// TwinCAT 3 PLC project Gemma
// ProgramVersion: 3.1.4024.0
// libraries:
//   CmpBitmapPool, * (System)
//   Tc2_Standard, * (Beckhoff Automation GmbH)
//   Tc2_System, * (Beckhoff Automation GmbH)
//   Tc3_Module, * (Beckhoff Automation GmbH)
//   VisuDialogs, * (System)
// project tree:
//   DUTs/ E_GEMMA.TcDUT (not stored)
//   / GlobalTextList.TcGTLO, PlcTask.TcTTO, Visualization Manager.TcVMO (not stored)
//   POUs/Estacion/ FB_Coordinador_SFC.TcPOU (not stored), FB_Director.TcPOU (not stored), FB_Estacion.TcPOU
//   POUs/ MAIN.TcPOU
//   POUs/Reloj/ FB_Clock.TcPOU (not stored)
//   POUs/Tareas/ FB_AlimentadorVerificadorDesplazador_SFC.TcPOU (not stored), FB_CheckMaterial_SFC.TcPOU (not stored), FB_Descargador_SFC.TcPOU (not stored), FB_EstacionFinalizar_SFC.TcPOU, FB_EstacionPreparar_SFC.TcPOU (not stored), FB_Rechazador_SFC.TcPOU, FB_ResetDescargador_SFC.TcPOU, FB_SituarPale_SFC.TcPOU (not stored), FB_TransferirPale_SFC.TcPOU
//   VISUs/ ImagePool.TcIPO (not stored), Visualization.TcVIS
// (motion and I/O tree: see PLC project manual)
// real-time tasks:
//   TASK PlcTask: cycle T#10ms, priority 20, ADS port 350
//   TASK PlcTask1: cycle T#10ms, priority 21, ADS port 351
// variable links:
//   Gemma/Gemma Instance <-> Device 1 (EtherCAT)/Term 1 (EK1200)/Term 2 (EL1008)
//     PlcTask Inputs/MAIN.Estacion.Codigo_pale_bit_0 <-> Channel 7/Codigo de palé bit 0
//     PlcTask Inputs/MAIN.Estacion.Codigo_pale_bit_1 <-> Channel 8/Codigo de palé bit 1
//     PlcTask Inputs/MAIN.Estacion.EstacionConectada <-> Channel 5/Parte operativa conectada (armada)
//     PlcTask Inputs/MAIN.Estacion.Presencia_pale <-> Channel 6/presencia de palé
//     PlcTask Inputs/MAIN.Estacion.Pulsador_marcha <-> Channel 3/Pulsador de marcha
//     PlcTask Inputs/MAIN.Estacion.Pulsador_parada_NC <-> Channel 4/Pulsador de parada [NC]
//     PlcTask Inputs/MAIN.Estacion.Pulsador_parada_emergencia <-> Channel 1/Pulsador de parada de emergencia
//     PlcTask Inputs/MAIN.Estacion.Selector_modo_manual <-> Channel 2/Selector de modo manual
//   Gemma/Gemma Instance <-> Device 1 (EtherCAT)/Term 1 (EK1200)/Term 3 (EL1008)
//     PlcTask Inputs/MAIN.Estacion.Codigo_pale_bit_2 <-> Channel 1/Código de palé bit 2
//     PlcTask Inputs/MAIN.Estacion.Detector_presion <-> Channel 2/Detector de presión
//   Gemma/Gemma Instance <-> Device 1 (EtherCAT)/Term 1 (EK1200)/Term 6 (EL1008)
//     PlcTask Inputs/MAIN.Estacion.Desplazador_detras <-> Channel 7/Cilindro del desplazador detrás
//     PlcTask Inputs/MAIN.Estacion.Horizontal_descargador_delante <-> Channel 2/Cilindro horizontal del descargador delante (sobre el palé)
//     PlcTask Inputs/MAIN.Estacion.Horizontal_descargador_detras <-> Channel 1/Cilindro horizontal del descargador detrás (sobre el punto de descarga)
//     PlcTask Inputs/MAIN.Estacion.Verificador_abajo <-> Channel 6/Cilindro del verificador abajo
//     PlcTask Inputs/MAIN.Estacion.Verificador_arriba <-> Channel 5/Cilindro del verificador arriba
//     PlcTask Inputs/MAIN.Estacion.Vertical_descargador_abajo <-> Channel 4/Cilindro vertical del descargador abajo
//     PlcTask Inputs/MAIN.Estacion.Vertical_descargador_arriba <-> Channel 3/Cilindro vertical del descargador arriba
//   Gemma/Gemma Instance <-> Device 1 (EtherCAT)/Term 1 (EK1200)/Term 7 (EL1008)
//     PlcTask Inputs/MAIN.Estacion.Base_en_alimentador <-> Channel 3/Presencia de base en el alimentador

CONFIGURATION Gemma
    RESOURCE PLC ON TwinCAT3
        TASK PlcTask(INTERVAL := T#10ms, PRIORITY := 20);
        PROGRAM MAIN WITH PlcTask : MAIN;
    END_RESOURCE
END_CONFIGURATION

// ---- POUs/MAIN.TcPOU
PROGRAM MAIN
VAR
	
	//Pulsador AT %I*: BOOL;
	//Lampara AT %Q*: BOOL;
	
	Estacion: FB_Estacion;

END_VAR

Estacion();

END_PROGRAM

// ---- POUs/Estacion/FB_Estacion.TcPOU
FUNCTION_BLOCK FB_Estacion
VAR_INPUT
    EstadoPausa: BOOL;
    EstadoReinicia: BOOL;
    CiclosSolicitados: UINT := 0;
    
    Tcheck: TIME := T#1S;
    Treset: TIME := T#1S;
    Tdesplazador: TIME := T#1S;
	Tcinta: TIME := T#0.5S;
END_VAR
VAR_OUTPUT
    CondicionInicial: BOOL := TRUE;
    CiclosPendientes: UINT;
    CiclosAceptados: UINT;
	CiclosRechazados: UINT;
    PaleCodigo: BYTE;
	pieza_ok: BOOL;
    
    // Entradas comunes
	Base_en_alimentador AT %I*: BOOL;
    Pulsador_parada_emergencia AT %I*: BOOL;
    Selector_modo_manual AT %I*: BOOL;
    Pulsador_marcha AT %I*: BOOL;
    Pulsador_parada_NC AT %I*: BOOL := TRUE; // Contacto normalmente cerrado
    EstacionConectada AT %I*: BOOL := TRUE;
    Detector_presion AT %I*: BOOL := TRUE;

    Presencia_pale AT %I*: BOOL;
    Codigo_pale_bit_0 AT %I*: BOOL;
    Codigo_pale_bit_1 AT %I*: BOOL;
    Codigo_pale_bit_2 AT %I*: BOOL;

    // Entradas espeficicas
    //Terminal 6
	Horizontal_descargador_detras AT %I*: BOOL;
	Horizontal_descargador_delante AT %I*: BOOL;
	Vertical_descargador_arriba AT %I*: BOOL;
	Vertical_descargador_abajo AT %I*: BOOL;
	Verificador_arriba AT %I*: BOOL;
	Verificador_abajo AT %I*: BOOL;
	Desplazador_detras AT %I*: BOOL;
	//Desplazador_delante AT %I*: BOOL;
	Alimentador_detras AT %I*: BOOL;
	
	
	//Terminal 7
	Alimentador_delante AT %I*: BOOL;
	Vacio_obtenido_vacuostato_descargador AT %I*: BOOL;

END_VAR
VAR
	ModoAnterior: E_GEMMA;    

    // Bloques funcionales
    CLK: FB_Clock;	

    // Bloques funcionales
	Director : FB_Director;
    Coordinador: FB_Coordinador_SFC;
	ChequeaMaterial: FB_CheckMaterial_SFC;
	AlimentadorVerificadorDesplazador: FB_AlimentadorVerificadorDesplazador_SFC;
    SituarPale: FB_SituarPale_SFC;
	ResetDescargador: FB_ResetDescargador_SFC;
    Descargador: FB_Descargador_SFC;
    Rechazador: FB_Rechazador_SFC;
    TransferirPale: FB_TransferirPale_SFC;
	Finalizar: FB_EstacionFinalizar_SFC;
	Preparar: FB_EstacionPreparar_SFC;
    
    // Salidas comunes
    Desconecta_parte_operativa AT %Q*: BOOL;
    Lampara_falta_material AT %Q*: BOOL;
    Lampara_marcha AT %Q*: BOOL;
    Lampara_alarma AT %Q*: BOOL;

    Activa_marcha_motor_cinta AT %Q*: BOOL;
    Invierte_marcha_motor_cinta AT %Q*: BOOL;
    Retenedor_pale_baja AT %Q*: BOOL;
    Separador_pale_sube AT %Q*: BOOL;
    
    //Terminal 8
	Descargador_adelante AT %Q*: BOOL;
	Descargador_atras AT %Q*: BOOL;
	Descargador_baja AT %Q*: BOOL;
	Rechazador_adelante AT %Q*: BOOL;
	Verificador_baja AT %Q*: BOOL;
	Desplazador_adelante AT %Q*: BOOL;
	Alimentador_adelante AT %Q*: BOOL;
	Eyector_succiona AT %Q*: BOOL;
	SFCPause: BOOL;
END_VAR

// Modo Automático
//IF NOT Selector_Modo_Manual THEN
CLK();

    // Bloques Funcionales
    Director(
        CondicionInicial := CondicionInicial,
        CondicionMarcha:= (CiclosSolicitados > 0) AND CondicionInicial,
        Emergencia := Pulsador_parada_emergencia,
        Finalizada := Finalizar.Done,
        FinTarea := (CiclosPendientes = 0),
        FinCiclo := Coordinador.Done,
        Manual := Selector_modo_manual,
        Marcha := Pulsador_marcha,
        ParaCiclo := NOT Pulsador_parada_NC,
        Preparada := Preparar.Done,
        Reinicia := EstadoReinicia
    );
	
	IF (Director.Modo <> E_GEMMA.F4) THEN

    SituarPale( //SituarPale
        SFCPause := NOT EstadoReinicia AND EstadoPausa,
        SFCReset := EstadoReinicia,
        Ack := NOT Coordinador.SituaPale,
        Execute := Coordinador.SituaPale,
        Tcinta := Tcinta,
        Presencia_pale := Presencia_pale,
           //Codigo_pale_bit_0 := Codigo_pale_bit_0,
        //Codigo_pale_bit_1 := Codigo_pale_bit_1,
        //Codigo_pale_bit_2 := Codigo_pale_bit_2

    );

	// Bloques Funcionales
	Coordinador(

		CiclosPendientes := CiclosPendientes,
		CiclosAceptados := CiclosAceptados,
		CiclosSolicitados := CiclosSolicitados,
		CiclosRechazados := CiclosRechazados,
		SFCPause := NOT EstadoReinicia AND EstadoPausa,
        SFCReset := EstadoReinicia,
		Ack := TRUE,
        Execute := (Director.Modo = E_GEMMA.F1),
		PaleSituado := SituarPale.Done,
		HayMaterial := ChequeaMaterial.Done,
		Verificado := AlimentadorVerificadorDesplazador.Done,
		DescargadorReseteado := ResetDescargador.Done,
        Rechazado := Rechazador.Done,
		BaseCargada := Descargador.Done,
		PaleTransferido := TransferirPale.Done,
		pieza_ok := pieza_ok
		
	);
	
	Preparar(
		
		SFCPause := NOT EstadoReinicia AND EstadoPausa,
        SFCReset := EstadoReinicia,
        Ack := (Director.Modo <> E_GEMMA.F2),
        Execute := (Director.Modo = E_GEMMA.F2),
		Horizontal_descargador_detras := Horizontal_descargador_detras,
		Vertical_descargador_arriba := Vertical_descargador_arriba,
		Presencia_pale := Presencia_pale
	
	);
	
	Finalizar(
		
		SFCPause := NOT EstadoReinicia AND EstadoPausa,
        SFCReset := EstadoReinicia,
        Ack := (Director.Modo <> E_GEMMA.F3),
        Execute := (Director.Modo = E_GEMMA.F3),
		Horizontal_descargador_detras := Horizontal_descargador_detras,
		Vertical_descargador_arriba := Vertical_descargador_arriba,
		Presencia_pale := Presencia_pale
	
	);
	
	SituarPale(

		SFCPause := NOT EstadoReinicia AND EstadoPausa,
        SFCReset := EstadoReinicia,
        Ack := NOT Coordinador.SituaPale,
        Execute := Coordinador.SituaPale,
        Tcinta := Tcinta,
        Presencia_pale := Presencia_pale,
       	//Codigo_pale_bit_0 := Codigo_pale_bit_0,
        //Codigo_pale_bit_1 := Codigo_pale_bit_1,
        //Codigo_pale_bit_2 := Codigo_pale_bit_2

	);
	
	ChequeaMaterial(
		Ack := NOT Coordinador.ChequeaMaterial,
		SFCPause := NOT EstadoReinicia AND EstadoPausa,
        SFCReset := EstadoReinicia,
		Execute := Coordinador.ChequeaMaterial,
		Base_en_Alimentador := Base_en_alimentador,
		Pulsador_marcha := Pulsador_marcha
	);
	
	AlimentadorVerificadorDesplazador(
		
		Ack := NOT Coordinador.VerificaBase,
        Tcheck := Tcheck,
		SFCPause := NOT EstadoReinicia AND EstadoPausa,
        SFCReset := EstadoReinicia,
		Execute := Coordinador.VerificaBase,
		Alimentador_delante := Alimentador_delante,
		Alimentador_detras := Alimentador_detras,
		Verificador_arriba := Verificador_arriba ,
		Verificador_abajo := Verificador_abajo,
		Desplazador_delante := Desplazador_delante,
		Desplazador_detras := Desplazador_detras, 
		
	);
	
	ResetDescargador(

		Ack := NOT Coordinador.ResetDescargador,
		SFCPause := NOT EstadoReinicia AND EstadoPausa,
        SFCReset := EstadoReinicia,
		Execute := Coordinador.ResetDescargador,
		Horizontal_descargador_detras := Horizontal_descargador_detras,
		Vertical_descargador_arriba := Vertical_descargador_arriba
	);
	
	Descargador(
		
		Ack := NOT Coordinador.CargaBase,
		SFCPause := NOT EstadoReinicia AND EstadoPausa,
        SFCReset := EstadoReinicia,
		Execute := Coordinador.CargaBase,
		Horizontal_descargador_detras := Horizontal_descargador_detras,
		Vertical_descargador_abajo := Vertical_descargador_abajo,
		Vacio_obtenido_vacuostato_descargador := Vacio_obtenido_vacuostato_descargador ,
		Vertical_descargador_arriba := Vertical_descargador_arriba ,
		Horizontal_descargador_delante := Horizontal_descargador_delante ,
	
	);	
		
	Rechazador(
		
		Ack := NOT Coordinador.RechazaBase,
		SFCPause := NOT EstadoReinicia AND EstadoPausa,
        SFCReset := EstadoReinicia,
		Execute := Coordinador.RechazaBase,
		Verificador_abajo := Verificador_abajo
		
	);
	
	TransferirPale(
	
		Ack := NOT Coordinador.TransfierePale,
		SFCPause := NOT EstadoReinicia AND EstadoPausa,
        SFCReset := EstadoReinicia,
		Execute := Coordinador.TransfierePale,

	);
	
	//Acciones Comunes
	// Parametros de Salida
	//Lampara_falta_material := ChequeaMaterial.Lampara_falta_material;
	Activa_marcha_motor_cinta := SituarPale.Activa_marcha_motor_cinta OR TransferirPale.Activa_marcha_motor_cinta OR Preparar.Activa_marcha_motor_cinta OR Finalizar.Activa_marcha_motor_cinta;
	//CheckMaterial
	Lampara_alarma := ChequeaMaterial.LamparaAlarma;
	Lampara_falta_material := ChequeaMaterial.Lampara_falta_material;
	//TranferirPale
	 Retenedor_pale_baja := TransferirPale.Retenedor_pale_baja;
	 Separador_pale_sube := TransferirPale.Separador_pale_sube;
	//AlimentadorVerificadorDesplazador
	Alimentador_adelante := AlimentadorVerificadorDesplazador.Alimentador_adelante;
	Verificador_baja := AlimentadorVerificadorDesplazador.Verificador_baja;
	Desplazador_adelante := AlimentadorVerificadorDesplazador.Desplazador_adelante;
	pieza_ok := AlimentadorVerificadorDesplazador.pieza_ok;
	//Descargador
	Eyector_succiona := Descargador.Eyector_succiona;
	Descargador_adelante := Descargador.Descargador_adelante;
	Descargador_atras := Descargador.Descargador_atras OR ResetDescargador.Descargador_atras;
	Descargador_baja := Descargador.Descargador_baja;
	//Rechazador
	Rechazador_adelante := Rechazador.Rechazador_adelante;
	
	IF NOT EstadoPausa THEN
	
		EstadoPausa := not Pulsador_parada_NC;
	
	ELSE
	
		EstadoPausa := NOT Pulsador_marcha;
	
	END_IF

END_IF	
	
// Parametros de Salida
CondicionInicial := EstacionConectada; //AND Desplazador_detras AND Verificador_arriba AND Vertical_descargador_arriba AND Alimentador_detras;

//al iniciar una tarea
IF ((ModoAnterior = E_GEMMA.A1) AND (Director.Modo <> E_GEMMA.A1) AND (CiclosPendientes = 0)) THEN
    CiclosPendientes := CiclosSolicitados;
END_IF

//IF (Director.Modo <> E_GEMMA.F4) THEN
    //PaleCodigo := SituarPale.PaleCodigo;
//ELSE 
    //PaleCodigo.0 := Codigo_pale_bit_0;
    //PaleCodigo.1 := Codigo_pale_bit_1;
    //PaleCodigo.2 := Codigo_pale_bit_2;
//END_IF

// ACTULIZACION DE IMAGENES
ModoAnterior := Director.Modo;

END_FUNCTION_BLOCK

// ---- POUs/Tareas/FB_ResetDescargador_SFC.TcPOU
FUNCTION_BLOCK FB_ResetDescargador_SFC

VAR_INPUT
	//nuestras_variables

    // SFC-Flags
    SFCPause: BOOL;
    SFCReset: BOOL;
    
    // Indicadores de sincronizacion
    Ack: BOOL := TRUE;
    Execute: BOOL;
	
	//Entradas
    Horizontal_descargador_detras: BOOL;
	Vertical_descargador_arriba: BOOL;

	
END_VAR
VAR_OUTPUT
    // Indicadores de sincronizacion
    Done: BOOL;
    Ready: BOOL;

	//Salidas
	Descargador_atras: BOOL;
	
END_VAR
VAR
END_VAR

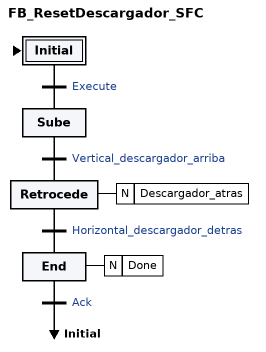
INITIAL_STEP Initial:
END_STEP
TRANSITION FROM Initial TO Sube
    := Execute;
END_TRANSITION
STEP Sube:
END_STEP
TRANSITION FROM Sube TO Retrocede
    := Vertical_descargador_arriba;
END_TRANSITION
STEP Retrocede:
    Descargador_atras(N);
END_STEP
TRANSITION FROM Retrocede TO End
    := Horizontal_descargador_detras;
END_TRANSITION
STEP End:
    Done(N);
END_STEP
TRANSITION FROM End TO Initial
    := Ack;
END_TRANSITION

END_FUNCTION_BLOCK

// ---- POUs/Tareas/FB_Rechazador_SFC.TcPOU
FUNCTION_BLOCK FB_Rechazador_SFC
VAR_INPUT
	
	//Tiempo
	Tcheck: TIME := T#1S;	

	// SFC-Flags
	SFCPause: BOOL;
	SFCReset: BOOL;
	
	//Indicadores de sincronizacion
	Ack: BOOL:= TRUE;
	Execute: BOOL;
	
	//Entradas
	
	Verificador_abajo: BOOL;

	
END_VAR
VAR_OUTPUT
	//indicadores de sincronizacion
	Done: BOOL;
	Ready: BOOL;

	//Salidas
	Rechazador_adelante: BOOL;
	
END_VAR
VAR
END_VAR

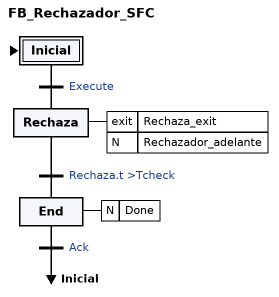
INITIAL_STEP Inicial:
END_STEP
TRANSITION FROM Inicial TO Rechaza
    := Execute;
END_TRANSITION
STEP Rechaza:
    Rechaza_exit(P0);  // exit action
    Rechazador_adelante(N);
END_STEP
TRANSITION FROM Rechaza TO End
    := Rechaza.t >Tcheck;
END_TRANSITION
STEP End:
    Done(N);
END_STEP
TRANSITION FROM End TO Inicial
    := Ack;
END_TRANSITION

ACTION Rechaza_exit:

END_ACTION

END_FUNCTION_BLOCK

// ---- POUs/Tareas/FB_TransferirPale_SFC.TcPOU
FUNCTION_BLOCK FB_TransferirPale_SFC
VAR_INPUT
	
	//Tiempo
	Tcheck: TIME := T#1S;	

	// SFC-Flags
	SFCPause: BOOL;
	SFCReset: BOOL;
	
	//Indicadores de sincronizacion
	Ack: BOOL:= TRUE;
	Execute: BOOL;
	
	//Entradas

	
END_VAR
VAR_OUTPUT
	//indicadores de sincronizacion
	Done: BOOL;
	Ready: BOOL;

	//Salidas
	Retenedor_pale_baja: BOOL;
	Activa_marcha_motor_cinta: BOOL;
	Separador_pale_sube: BOOL;
	
END_VAR
VAR
END_VAR

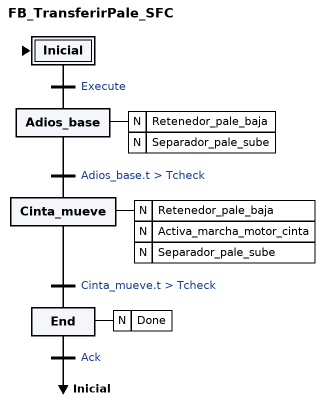
INITIAL_STEP Inicial:
END_STEP
TRANSITION FROM Inicial TO Adios_base
    := Execute;
END_TRANSITION
STEP Adios_base:
    Retenedor_pale_baja(N);
    Separador_pale_sube(N);
END_STEP
TRANSITION FROM Adios_base TO Cinta_mueve
    := Adios_base.t > Tcheck;
END_TRANSITION
STEP Cinta_mueve:
    Retenedor_pale_baja(N);
    Activa_marcha_motor_cinta(N);
    Separador_pale_sube(N);
END_STEP
TRANSITION FROM Cinta_mueve TO End
    := Cinta_mueve.t > Tcheck;
END_TRANSITION
STEP End:
    Done(N);
END_STEP
TRANSITION FROM End TO Inicial
    := Ack;
END_TRANSITION

END_FUNCTION_BLOCK

// ---- POUs/Tareas/FB_EstacionFinalizar_SFC.TcPOU
FUNCTION_BLOCK FB_EstacionFinalizar_SFC
VAR_INPUT
	//nuestras_variables
	Tcinta: TIME := T#0.5S;	

    // SFC-Flags
    SFCPause: BOOL;
    SFCReset: BOOL;

    // Indicadores de sincronizacion
    Ack: BOOL := TRUE;
    Execute: BOOL;

   //Entradas
    Horizontal_descargador_detras: BOOL;
	Vertical_descargador_arriba: BOOL;
	Presencia_pale: BOOL;
	
END_VAR
VAR_OUTPUT
    // Indicadores de sincronizacion
    Done: BOOL;
    Ready: BOOL;
	
	//Salidas
	Descargador_atras: BOOL;
	Activa_marcha_motor_cinta: BOOL;
END_VAR
VAR
	Tcinta: TIME := T#0.5S;
END_VAR

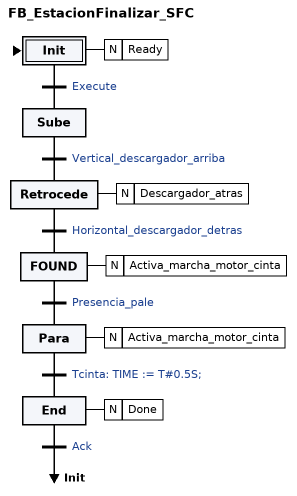
INITIAL_STEP Init:
    Ready(N);
END_STEP
TRANSITION FROM Init TO Sube
    := Execute;
END_TRANSITION
STEP Sube:
END_STEP
TRANSITION FROM Sube TO Retrocede
    := Vertical_descargador_arriba;
END_TRANSITION
STEP Retrocede:
    Descargador_atras(N);
END_STEP
TRANSITION FROM Retrocede TO FOUND
    := Horizontal_descargador_detras;
END_TRANSITION
STEP FOUND:
    Activa_marcha_motor_cinta(N);
END_STEP
TRANSITION FROM FOUND TO Para
    := Presencia_pale;
END_TRANSITION
STEP Para:
    Activa_marcha_motor_cinta(N);
END_STEP
TRANSITION FROM Para TO End
    := Tcinta: TIME := T#0.5S;
END_TRANSITION
STEP End:
    Done(N);
END_STEP
TRANSITION FROM End TO Init
    := Ack;
END_TRANSITION

END_FUNCTION_BLOCK

// ---- GlobalTextList.TcGTLO
TEXTLIST GlobalTextList
  189 = '  ➡ ⬅ ⬇ ⬆ ← → ↓ ↑'
  198 = ' ➙'
  307 = '%i'
  611 = '0'
  472 = '1'
  731 = '<'
  44 = '>'
  12 = 'A+'
  482 = 'A-'
  789 = 'Abajo'
  231 = 'Aceptados'
  66 = 'Alarma'
  224 = 'Alimentador'
  25 = 'Arriba'
  54 = 'Aspirar'
  267 = 'B+'
  782 = 'B-'
  801 = 'C+'
  215 = 'C-'
  701 = 'Ciclos'
  642 = 'Ciclos Completados'
  957 = 'Cinta'
  81 = 'Colocado'
  497 = 'Comenzar'
  143 = 'D+'
  630 = 'D-'
  481 = 'Delante'
  437 = 'Descargador'
  936 = 'Desplazador'
  445 = 'Detrás'
  74 = 'E+'
  781 = 'E-'
  742 = 'E-Stop'
  908 = 'Estado'
  286 = 'Estoy Abajo'
  148 = 'Estoy Arriba'
  955 = 'Eyector'
  417 = 'F+'
  707 = 'F-'
  878 = 'FALTA M.'
  395 = 'FM'
  769 = 'FMS-201                                 ALIMENTADORA DE BASES                                                    VTL     '
  561 = 'Horizontal'
  750 = 'Lámpara'
  45 = 'Marcha'
  634 = 'Material'
  861 = 'Panel'
  463 = 'Parada'
  708 = 'Pausa'
  619 = 'pb'
  935 = 'Pieza NO OK'
  336 = 'Pieza OK'
  741 = 'Pieza Ok'
  524 = 'Planta'
  640 = 'pp'
  783 = 'Preparado'
  330 = 'R+'
  876 = 'Rechazador'
  970 = 'Rechazados'
  888 = 'Rechazads'
  94 = 'Rehczados'
  614 = 'Reset'
  560 = 'Restantes'
  531 = 'Rev'
  452 = 'Run'
  784 = 'S+'
  918 = 'Solicitados'
  815 = 'Succionar'
  643 = 'Tarea'
  710 = 'V+'
  288 = 'V-'
  629 = 'Vacío'
  125 = 'Verificador'
  839 = 'Verificador Activado'
  483 = 'Vertical'
  575 = '➡'
  509 = '⬅'
  381 = '⬆'
  169 = '⬇'
END_TEXTLIST

// ---- VISUs/Visualization.TcVIS
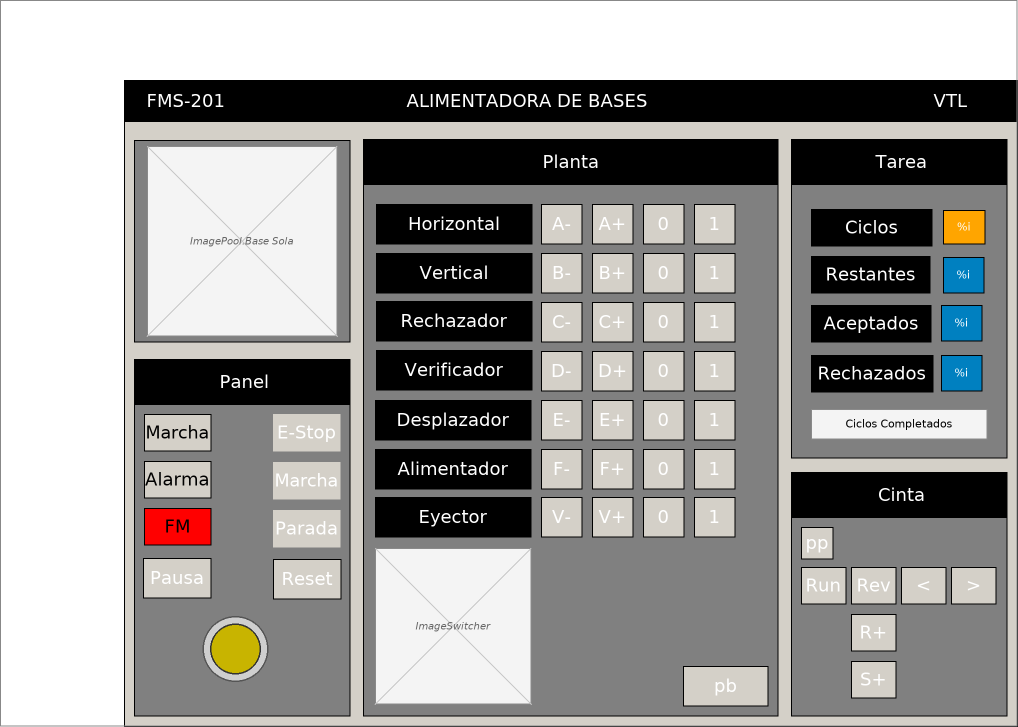
VISUALIZATION Visualization  // 1018x727
    Rectangle (124,121 894x606)
    Rectangle (791,184 216x274)
    Rectangle (363,184 415x532)
    Rectangle (363,139 415x45)
    Label (363,141 416x42), "Planta"
    Rectangle (791,139 216x45)
    Label (841,144 121x36), "Tarea"
    Progressbar (811,409 176x30), "Ciclos Completados", variable: MAIN.test_pieza.Aceptados
    RoundedRectangle (376,204 156x40), "Horizontal"
    Textfield (943,210 42x34), "%i", text variable: MAIN.Estacion.CiclosSolicitados
        OnMouseDown: write MAIN.Estacion.CiclosSolicitados via VisuDialogs.Numpad, min 1, max 10
    RoundedRectangle (811,209 121x37), "Ciclos"
    RoundedRectangle (811,256 119x37), "Restantes"
    RoundedRectangle (811,305 120x37), "Aceptados"
    RoundedRectangle (811,355 122x37), "Rechazados"
    Textfield (943,257 41x36), "%i", text variable: MAIN.Estacion.CiclosPendientes
    Textfield (941,305 41x36), "%i", text variable: MAIN.Estacion.CiclosAceptados
    Textfield (941,355 41x36), "%i", text variable: MAIN.Estacion.CiclosRechazados
    RoundedRectangle (592,253 41x40), "B+", colour toggle: MAIN.Estacion.Descargador_baja
        toggle MAIN.Estacion.Descargador_baja
    Rectangle (791,517 216x199)
    Rectangle (791,472 216x45)
    Label (841,477 121x36), "Cinta"
    Rectangle (134,140 216x202)
    Rectangle (134,404 216x312)
    Rectangle (134,359 216x45)
    Label (184,364 121x36), "Panel"
    Rectangle (124,80 894x41)
    Label (124,81 893x40), "FMS-201 ALIMENTADORA DE BASES VTL"
    RoundedRectangle (376,253 156x40), "Vertical"
    RoundedRectangle (592,204 41x40), "A+", colour toggle: MAIN.Estacion.Descargador_adelante
        tap MAIN.Estacion.Descargador_adelante
    RoundedRectangle (592,302 41x40), "C+", colour toggle: MAIN.Estacion.Rechazador_adelante
        tap MAIN.Estacion.Rechazador_adelante
    RoundedRectangle (592,351 41x40), "D+", colour toggle: MAIN.Estacion.Verificador_baja
        tap MAIN.Estacion.Verificador_baja
    RoundedRectangle (592,400 41x40), "E+", colour toggle: MAIN.Estacion.Desplazador_adelante
        tap MAIN.Estacion.Desplazador_adelante
    RoundedRectangle (592,449 41x40), "F+", colour toggle: MAIN.Estacion.Alimentador_adelante
        tap MAIN.Estacion.Alimentador_adelante
    RoundedRectangle (592,497 41x40), "V+", colour toggle: MAIN.Estacion.Eyector_succiona
        toggle MAIN.Estacion.Eyector_succiona
    RoundedRectangle (376,301 156x40), "Rechazador"
    RoundedRectangle (376,350 156x40), "Verificador"
    RoundedRectangle (375,400 156x40), "Desplazador"
    RoundedRectangle (375,449 156x40), "Alimentador"
    RoundedRectangle (375,497 156x40), "Eyector"
    RoundedRectangle (541,204 41x40), "A-", colour toggle: MAIN.Estacion.Descargador_atras
        tap MAIN.Estacion.Descargador_atras
    RoundedRectangle (643,204 41x40), "0", colour toggle: MAIN.Estacion.Horizontal_descargador_detras
    RoundedRectangle (694,204 41x40), "1", colour toggle: MAIN.Estacion.Horizontal_descargador_delante
    RoundedRectangle (643,253 41x40), "0", colour toggle: MAIN.Estacion.Vertical_descargador_arriba
        tap MAIN.Estacion.Vertical_descargador_arriba
    RoundedRectangle (694,253 41x40), "1", colour toggle: MAIN.Estacion.Vertical_descargador_abajo
        tap MAIN.Estacion.Vertical_descargador_abajo
    RoundedRectangle (643,302 41x40), "0"
    RoundedRectangle (643,351 41x40), "0", colour toggle: MAIN.Estacion.Verificador_arriba
        tap MAIN.Estacion.Verificador_arriba
    RoundedRectangle (643,400 41x40), "0", colour toggle: MAIN.Estacion.Desplazador_detras
        tap MAIN.Estacion.Desplazador_detras
    RoundedRectangle (643,449 41x40), "0", colour toggle: MAIN.Estacion.Alimentador_detras
        tap MAIN.Estacion.Alimentador_detras
    RoundedRectangle (643,497 41x40), "0"
    RoundedRectangle (694,302 41x40), "1"
    RoundedRectangle (694,351 41x40), "1", colour toggle: MAIN.Estacion.Verificador_abajo
        tap MAIN.Estacion.Verificador_abajo
    RoundedRectangle (694,400 41x40), "1"
    RoundedRectangle (694,449 41x40), "1", colour toggle: MAIN.Estacion.Alimentador_delante
        tap MAIN.Estacion.Alimentador_delante
    RoundedRectangle (694,497 41x40), "1", colour toggle: MAIN.Estacion.Vacio_obtenido_vacuostato_descargador
        tap MAIN.Estacion.Vacio_obtenido_vacuostato_descargador
    RoundedRectangle (541,253 41x40), "B-"
    RoundedRectangle (541,302 41x40), "C-"
    RoundedRectangle (541,351 41x40), "D-"
    RoundedRectangle (541,400 41x40), "E-"
    RoundedRectangle (541,449 41x40), "F-"
    RoundedRectangle (541,497 41x40), "V-"
    RoundedRectangle (683,666 85x40), "pb", colour toggle: MAIN.Estacion.Base_en_Alimentador
        tap MAIN.Estacion.Base_en_Alimentador
    RoundedRectangle (144,508 67x37), "FM", colour toggle: MAIN.Estacion.Lampara_falta_material
        tap MAIN.Estacion.Lampara_falta_material
    RoundedRectangle (801,527 32x32), "pp", colour toggle: MAIN.Estacion.Presencia_pale
        tap MAIN.Estacion.Presencia_pale
    RoundedRectangle (951,567 45x37), ">", colour toggle: MAIN.Estacion.Activa_marcha_motor_cinta
        tap MAIN.Estacion.Activa_marcha_motor_cinta
    RoundedRectangle (901,567 45x37), "<", colour toggle: MAIN.Estacion.Invierte_marcha_motor_cinta
        toggle MAIN.Estacion.Invierte_marcha_motor_cinta
    RoundedRectangle (801,567 45x37), "Run", colour toggle: MAIN.Estacion.Activa_marcha_motor_cinta
    RoundedRectangle (851,567 45x37), "Rev", colour toggle: MAIN.Estacion.Invierte_marcha_motor_cinta
    RoundedRectangle (851,614 45x37), "R+", colour toggle: MAIN.Estacion.Retenedor_pale_baja
        toggle MAIN.Estacion.Retenedor_pale_baja
    RoundedRectangle (851,661 45x37), "S+", colour toggle: MAIN.Estacion.Separador_pale_sube
        toggle MAIN.Estacion.Separador_pale_sube
    RoundedRectangle (273,414 67x37), "E-Stop", colour toggle: MAIN.Estacion.Pulsador_parada_emergencia
        tap MAIN.Estacion.Pulsador_parada_emergencia
    RoundedRectangle (273,462 67x37), "Marcha", colour toggle: MAIN.Estacion.Pulsador_marcha
        tap MAIN.Estacion.Pulsador_marcha
    RoundedRectangle (273,510 67x37), "Parada", colour toggle: MAIN.Estacion.Pulsador_parada_NC
        tap MAIN.Estacion.Pulsador_parada_NC
    RoundedRectangle (144,461 67x37), "Alarma", colour toggle: MAIN.Estacion.Lampara_alarma
        tap MAIN.Estacion.Lampara_alarma
    RoundedRectangle (144,414 67x37), "Marcha", colour toggle: MAIN.Estacion.Lampara_marcha
        tap MAIN.Estacion.Lampara_marcha
    Image (147,146 190x190), image: ImagePool.Base Sola
    Lamp1 (197,611 77x76), variable: MAIN.test_pieza.Lampara_falta_material, style: Lamp-Lamp1-Yellow
    ImageSwitcher (375,548 156x156), variable: MAIN.Estacion.pieza_ok, background image: ImagePool.Base OK, image: ImagePool.Base No OK, behaviour: TOGGLE
    RoundedRectangle (143,558 68x40), "Pausa", text variable: MAIN.Estacion.EstadoPausa, colour toggle: MAIN.Estacion.EstadoPausaMAIN.Estacion.EstadoPausa
        tap MAIN.Estacion.EstadoPausa
    RoundedRectangle (273,559 68x40), "Reset", text variable: MAIN.Estacion.EstadoReinicia, colour toggle: MAIN.Estacion.EstadoReinicia
        tap MAIN.Estacion.EstadoReinicia
END_VISUALIZATION
